FUNCTION_BLOCK AxesReset_Body EXTENDS Body_Task_Base
VAR_INPUT
END_VAR
VAR_OUTPUT
END_VAR
VAR
	resetMover : Tc2_MC2.MC_Reset;
	_axis : REFERENCE TO Tc2_MC2.AXIS_REF;
	_ResetMover : BOOL;
	state : INT;

END_VAR

CASE State OF
	0:
		IF _ResetMover THEN
			_done := FALSE;
			_error := FALSE;
			_busy := TRUE;
			resetMover.Execute := TRUE;
			IF resetMover.Busy THEN
				State := 10;
				_ResetMover := FALSE;
			END_IF
		END_IF
	
	10:
		IF NOT resetMover.Busy THEN
			IF resetMover.Done THEN
				_done := TRUE;
			ELSIF resetMover.Error THEN
				_error := TRUE;
			END_IF
			_busy := FALSE;
			resetMover.Execute := FALSE;
			State := 0;
		END_IF
END_CASE

resetMover(Axis := _axis);

METHOD Abort : BOOL
resetMover.Execute := FALSE;
_busy := FALSE;
_ResetMover := FALSE;
Abort := TRUE;
State := 0;
END_METHOD

PROPERTY Busy : BOOL
GET
Busy := _busy;
END_GET
END_PROPERTY

PROPERTY Done : BOOL
GET
Done := _done;
END_GET
END_PROPERTY

PROPERTY Error : BOOL
GET
Error := _error;
END_GET
END_PROPERTY

METHOD Execute : BOOL
VAR_INPUT
END_VAR
Execute := _ResetMover := true;
END_METHOD

METHOD FB_init : BOOL
VAR_INPUT
	bInitRetains : BOOL; // if TRUE, the retain variables are initialized (warm start / cold start)
	bInCopyCode : BOOL;  // if TRUE, the instance afterwards gets moved into the copy code (online change)
	axis : reference TO AXIS_REF;
END_VAR
_axis REF= axis;
END_METHOD

END_FUNCTION_BLOCK

(* stored: Version 1.1.0.1, ProductVersion 3.1.4024.11
   POU AxesReset_Body: Id {50b6cb56-c29b-4e65-9645-432ca640e140}, SpecialFunc None
   Method Abort: Id {1e191aa0-5300-47ad-a5cc-fd578ced08bc}
   Property Busy: Id {ffbd0dda-3106-42ba-b22c-3278cb6aaea4}
   Get Get: Id {90c7b31c-76e8-4f44-95af-c4317569bbe0}
   Property Done: Id {47e63658-753a-4115-96e1-42e82c8ff57f}
   Get Get: Id {accb34dd-8a4d-4cb7-bc9f-4596b11ba7cc}
   Property Error: Id {44b7813b-391c-4b03-b5bd-f887814b2c5c}
   Get Get: Id {e407d0a0-d259-4518-9091-03bbe8cf3bbe}
   Method Execute: Id {6a1f36ad-1cf4-4393-9c94-06ccb247a97f}
   Method FB_init: Id {8a85576b-5504-487e-903b-6d992319f896} *)
